FUNCTION_BLOCK Stopped_State  IMPLEMENTS ITF_State
VAR_INPUT
END_VAR
VAR_OUTPUT
END_VAR
VAR
	_state : ITF_PMLBase;
	_stateMachine : IPmlStateMachine;
END_VAR

METHOD Cycle : BOOL
VAR_INPUT
END_VAR
END_METHOD

METHOD FB_init : BOOL
VAR_INPUT
	bInitRetains : BOOL; // if TRUE, the retain variables are initialized (warm start / cold start)
	bInCopyCode : BOOL;  // if TRUE, the instance afterwards gets moved into the copy code (online change)
		state : ITF_PMLBase;
	statemachine : IPmlStateMachine;
END_VAR
_stateMachine := statemachine;
_state := state;
END_METHOD

END_FUNCTION_BLOCK

(* stored: Version 1.1.0.1, ProductVersion 3.1.4024.11
   POU Stopped_State: Id {07f75b01-2ab4-46f8-9e04-8a2d11283c1e}, SpecialFunc None
   Method Cycle: Id {089743e0-2e35-4480-914e-6129f9c4ab64}
   Method FB_init: Id {c4cc0871-9569-4d59-b9f4-6bd827de56f5} *)
